# EPICS StreamDevice protocol: U2021XASup/devU2021XA.proto
InTerminator = CR LF;

getTracTime{    out "getTracTime"; in "%f"; }

getTracData{
    ReplyTimeout=5000; ReadTimeout=100; Separator=", ";
                out "getTracData"; in "[%e]" }

getInstrInfo{   out "getInstrInfo"; in "%s"; }

getResources{   out "getResources"; in "%s"; }

setTracTime{ out "setTracTime %f"; in "%f"; }

query{ out "query \$1"; in "%s"; }
write{ out "write \$1"; in "%s"; }

instrConnect{    out "instrConnect";    in "%s"; }
instrDisconnect{ out "instrDisconnect"; in "%s"; }
instrInit{       out "instrInit";       in "%s"; }

debug{ out "%s"; in "%s"; }
